// TwinCAT 3 PLC project ApicoPLC
// ProgramVersion: 3.1.4023.0
// libraries:
//   SPT Base Types, * (Beckhoff Automation LLC)
//   SPT Components, * (Beckhoff Automation LLC)
//   SPT Event Logger, * (Beckhoff Automation LLC)
//   SPT Utilities, * (Beckhoff Automation LLC)
//   Tc2_EtherCAT, * (Beckhoff Automation GmbH)
//   Tc2_Standard, * (Beckhoff Automation GmbH)
//   Tc2_System, * (Beckhoff Automation GmbH)
//   Tc3_EventLogger, * (Beckhoff Automation GmbH)
//   Tc3_Module, * (Beckhoff Automation GmbH)
//   Tc3_PackML_V2, * (Beckhoff Automation GmbH)
//   VisuDialogs, * (System)
//   VisuSymbols,newest,System
// project tree:
//   DUTs/Recipe/ ST_AxisRecipe.TcDUT (not stored), ST_PullWheelsRecipe.TcDUT (not stored), ST_SealerRecipe.TcDUT (not stored), ST_UnwindRecipe.TcDUT (not stored)
//   DUTs/ ST_Descriptor2.TcDUT (not stored), ST_PackML_Control.TcDUT (not stored), ST_PackML_Control_Simplified.TcDUT (not stored)
//   / GlobalTextList.TcGTLO, MAIN.TcPOU, PlcTask.TcTTO (not stored), VisualizationManager.TcVMO (not stored)
//   Machine/Components/Cylinder/ FB_Cylinder.TcPOU (not stored), I_Cylinder.TcIO (not stored), ST_Cylinder_Command.TcDUT (not stored), ST_Cylinder_Config.TcDUT (not stored), ST_Cylinder_HMI.TcDUT (not stored), ST_Cylinder_Status.TcDUT (not stored)
//   Machine/Components/ FB_SealBar.TcPOU (not stored)
//   Machine/EquipmentModules/ FB_PullWheel.TcPOU, FB_Unwind.TcPOU (not stored), FB_Sealer.TcPOU (not stored)
//   Machine/ FB_Machine.TcPOU
//   Machine/HMI Connections/ FB_ControlSource_HMI.TcPOU (not stored), FB_ControlSource_HMI_Machine.TcPOU
//   Machine/Templates/ FB_EquipmentModuleTemplate.TcPOU (not stored)
//   Machine/VISUs/VisuOjects/ V_MachineModule.TcVIS (not stored), V_Module.TcVIS (not stored)
//   Machine/VISUs/ V_Main.TcVIS
// real-time tasks:
//   TASK PlcTask: cycle T#10ms, priority 20, ADS port 350
// motion (NC):
//   TASK NC-Task 1 SAF: cycle T#2ms, priority 4, ADS port 501
//   TASK NC-Task 1 SVB: cycle T#10ms, priority 8, ADS port 511
//   AXIS Unwind (id 4)
//   AXIS Seal (id 5)
//   AXIS Pull 1 (id 6)
//   AXIS Pull 2 (id 7)
// variable links:
//   ApicoPLC/ApicoPLC Instance <-> NC-Task 1 SAF/Axes/Pull 1
//     PlcTask Inputs/MAIN.ApicoSeed.PullWheels.LeftPullWheel.BasicSlaveAxis._Axis.NcToPlc <-> Outputs/ToPlc
//     PlcTask Outputs/MAIN.ApicoSeed.PullWheels.LeftPullWheel.BasicSlaveAxis._Axis.PlcToNc <-> Inputs/FromPlc
//   ApicoPLC/ApicoPLC Instance <-> NC-Task 1 SAF/Axes/Pull 2
//     PlcTask Inputs/MAIN.ApicoSeed.PullWheels.RightPullWheel.BasicSlaveAxis._Axis.NcToPlc <-> Outputs/ToPlc
//     PlcTask Outputs/MAIN.ApicoSeed.PullWheels.RightPullWheel.BasicSlaveAxis._Axis.PlcToNc <-> Inputs/FromPlc
//   ApicoPLC/ApicoPLC Instance <-> NC-Task 1 SAF/Axes/Seal
//     PlcTask Inputs/MAIN.ApicoSeed.Sealer.SealerAxis.BasicAxis._Axis.NcToPlc <-> Outputs/ToPlc
//     PlcTask Outputs/MAIN.ApicoSeed.Sealer.SealerAxis.BasicAxis._Axis.PlcToNc <-> Inputs/FromPlc
//   ApicoPLC/ApicoPLC Instance <-> NC-Task 1 SAF/Axes/Unwind
//     PlcTask Inputs/MAIN.ApicoSeed.Unwind.Axis.BasicAxis._Axis.NcToPlc <-> Outputs/ToPlc
//     PlcTask Outputs/MAIN.ApicoSeed.Unwind.Axis.BasicAxis._Axis.PlcToNc <-> Inputs/FromPlc

// ---- Machine/EquipmentModules/FB_PullWheel.TcPOU
FUNCTION_BLOCK FB_PullWheel EXTENDS FB_PackML_BaseModule
VAR
    // Sub module definitions here

    // List of sub modules
    ipSubModules_Init : ARRAY[1..Parameters_PackML_Base.MAX_NO_OF_SUBMODULES] OF I_PackML_BaseModule := [];

    // Component definitions here
    LeftPullWheel     : FB_Component_BasicSlaveAxis := (Name := 'Left');
    RightPullWheel    : FB_Component_BasicSlaveAxis := (Name := 'Right');
    PullWheelCylinder : FB_Cylinder                 := (Name := 'Cylinder');

    // List of Components
    ipComponents_Init : ARRAY[1..Parameters_PackML_Base.MAX_NO_OF_COMPONENTS] OF I_ComponentBase
        := [LeftPullWheel, RightPullWheel, PullWheelCylinder];

    //Alarms for this module
    PullWheelAlarms : ARRAY[1..PULL_WHEELS_ALARM_COUNT] OF FB_TcAlarm;

	//Data for recipe
	Recipe : ST_PullWheelsRecipe;
    (*Parameters from PackTags for module
    _Param  : ARRAY[1..10] OF ST_Descriptor2;*)
    _Report : ARRAY[1..10] OF ST_Descriptor2;

    //HMI Control for EM
    fbControlSourceHMI : FB_ControlSource_HMI;
END_VAR

VAR CONSTANT

    //reports 
    FAULT : INT := 1;

    //Alarms
    PULL_WHEELS_ALARM_COUNT : INT := 5;
END_VAR

//Simulation variables for messaging
VAR
    ErrorInput : BOOL;
    WarnInput  : BOOL;
    InfoInput  : BOOL;
END_VAR

METHOD PROTECTED Aborting
VAR_INPUT
END_VAR
CASE SequenceState OF
    0:
        NoStateTasksToComplete := FALSE;
        SequenceState          := SequenceState + 10;
    10:
        LeftPullWheel.Stop();
        RightPullWheel.Stop();
        IF LeftPullWheel.Stopped AND RightPullWheel.Stopped THEN
            SequenceState := SequenceState + 10;
        END_IF
    20:
        // Disable here
        LeftPullWheel.Disable();
        RightPullWheel.Disable();
        PullWheelCylinder.Retract();

        // Check not enabled here
        IF NOT LeftPullWheel.Enabled AND NOT RightPullWheel.Enabled AND PullWheelCylinder.Retracted THEN
            SequenceState := SequenceState + 10;
        END_IF

        StateTasksComplete := TRUE;
END_CASE

SUPER^.Aborting();
END_METHOD

PROPERTY Acceleration : LREAL
SET
Recipe.LeftAxis.Acceleration := Acceleration;
Recipe.RightAxis.Acceleration := Acceleration;
END_SET
END_PROPERTY

METHOD PROTECTED Clearing
VAR_INPUT
END_VAR
CASE SequenceState OF
    0:
        NoStateTasksToComplete := FALSE;
        SequenceState          := SequenceState + 10;
    10:
        //Reset any alarms that get latched
        PullWheelAlarms[E_PullWheels.StartTimeout].Clear(0, 0);
        SequenceState := SequenceState + 10;
    20:
        // Enable here
        LeftPullWheel.Enable();
        RightPullWheel.Enable();

        // Check enabled here
        IF LeftPullWheel.Enabled AND RightPullWheel.Enabled THEN
            SequenceState := SequenceState + 10;
        END_IF
    30:
        StateTasksComplete := TRUE;
END_CASE

SUPER^.Clearing();
END_METHOD

METHOD PROTECTED CreateEvents
VAR_INPUT
END_VAR
// Add your event creation here
F_CreateAllEventsInClass(Alarms     := PullWheelAlarms,
                         ClassSize  := SIZEOF(TC_EVENTS.PullWheels),
                         pInitEvent := ADR(TC_EVENTS.PullWheels.InitReferenceEvent),
                         Prefix     := _Name);

// Super call to base
SUPER^.CreateEvents();
END_METHOD

METHOD CyclicLogic
VAR_INPUT
END_VAR
IF NOT _InitComplete THEN
    _InitComplete := Initialize();
    RETURN;
END_IF

SUPER^.CyclicLogic();

//HMI control for EM
fbControlSourceHMI.CyclicLogic();

//Set the current alarm severity for this module
_CurrentAlarmSeverity := F_GetMaxSeverityRaised(Alarms := PullWheelAlarms, CurrentSeverity := _CurrentAlarmSeverity);

//Simulate Alarm Messaging
CyclicLogic_Simulation();
END_METHOD

METHOD CyclicLogic_Simulation
VAR_INPUT
END_VAR

VAR_INST
END_VAR
(*	
This is just for testing. Real hardware can be setup in other places
Here the alarms will raise and clear on its own if the input changes	
*)

//Generic Alarms for Testing
IF ErrorInput AND NOT PullWheelAlarms[E_PullWheels.AlarmMessage].bRaised THEN
    RaiseAlarm2Args(PullWheelAlarms[E_PullWheels.AlarmMessage], '', '');
ELSIF NOT ErrorInput AND PullWheelAlarms[E_PullWheels.AlarmMessage].bRaised THEN
    PullWheelAlarms[E_PullWheels.AlarmMessage].Clear(0, 0);
END_IF

IF WarnInput AND NOT PullWheelAlarms[E_PullWheels.WarnMessage].bRaised THEN
    RaiseAlarm2Args(PullWheelAlarms[E_PullWheels.WarnMessage], '', '');
ELSIF NOT WarnInput AND PullWheelAlarms[E_PullWheels.WarnMessage].bRaised THEN
    PullWheelAlarms[E_PullWheels.WarnMessage].Clear(0, 0);
END_IF

IF InfoInput AND NOT PullWheelAlarms[E_PullWheels.InfoMessage].bRaised THEN
    RaiseAlarm2Args(PullWheelAlarms[E_PullWheels.InfoMessage], '', '');
ELSIF NOT InfoInput AND PullWheelAlarms[E_PullWheels.InfoMessage].bRaised THEN
    PullWheelAlarms[E_PullWheels.InfoMessage].Clear(0, 0);
END_IF
END_METHOD

METHOD PROTECTED Execute
VAR_INPUT
END_VAR
// Function based on mode.  NO need to make SUPER^.Executing() since it does nothing.
CASE _CurrentMode OF
    E_PMLUnitMode.ePMLUnitMode_Production:
        IF LeftPullWheel.InPosition AND NOT LeftPullWheel.Busy THEN
            PullWheelCylinder.Retract();
            IF PullWheelCylinder.Retracted THEN
                StateComplete();
            END_IF
        END_IF
    E_PMLUnitMode.ePMLUnitMode_Maintenance:
        ;
    E_PMLUnitMode.ePMLUnitMode_Manual:
        ;
END_CASE
END_METHOD

//! @summary Basic module initialization logic
METHOD PROTECTED Initialize : BOOL;
VAR
    i                        : UDINT;
    varInfo                  : __SYSTEM.VAR_INFO;
    AllSubUnitsInitialized   : BOOL := TRUE;
    AllComponentsInitialized : BOOL := TRUE;
END_VAR

//! @description This method is called by <c>CyclicLogic()</c> as required
Initialize := FALSE;
CASE DescendantSequenceState OF
    0:
        // Define the interfaces to the different subunits (Must take place before SUPER^.initialize call)
        FOR i := 1 TO SPT_BaseTypes.Parameters_PackML_Base.MAX_NO_OF_SUBMODULES DO
            ipSubModules[i] := ipSubModules_Init[i];
        END_FOR

        FOR i := 1 TO SPT_BaseTypes.Parameters_PackML_Base.MAX_NO_OF_COMPONENTS DO
            ipComponents[i] := ipComponents_Init[i];
        END_FOR

        _LogModeChanges         := FALSE;
        _LogStateChanges        := FALSE;
        DescendantSequenceState := DescendantSequenceState + 10;
    10:
        //Setup Custom modes here

        (*CustomModes(eMode                          :=,
                    sName                          :=,
                    bDisableClearing               :=,
                    bDisableStarting               :=,
                    bDisableSuspended              :=,
                    bDisableStopping               :=,
                    bDisableAborting               :=,
                    bDisableHolding                :=,
                    bDisableHeld                   :=,
                    bDisableUnholding              :=,
                    bDisableSuspending             :=,
                    bDisableUnsuspending           :=,
                    bDisableResetting              :=,
                    bDisableIdle                   :=,
                    bDisableCompleting             :=,
                    bDisableComplete               :=,
                    bEnableUnitModeChangeStopped   :=,
                    bEnableUnitModeChangeIdle      :=,
                    bEnableUnitModeChangeSuspended :=,
                    bEnableUnitModeChangeExecute   :=,
                    bEnableUnitModeChangeAborted   :=,
                    bEnableUnitModeChangeHeld      :=,
                    bEnableUnitModeChangeComplete  :=,
                    bError                         =>,
                    nErrorId                       =>);*)
        DescendantSequenceState := DescendantSequenceState + 10;
    20:
        //Copy Mode names
        FOR i := 1 TO 3 DO
            ModeNames[i] := F_UnitModeToString(UDINT_TO_DINT(i));
        END_FOR

        Initialize_TagData();
		RegisterExternalController(Controller := fbControlSourceHMI);
		fbControlSourceHMI.CyclicLogic();
        DescendantSequenceState := DescendantSequenceState + 10;
    30:
        //Call the Super
        IF SUPER^.Initialize() THEN
            DescendantSequenceState := DescendantSequenceState + 10;
        END_IF
    40:
        Initialize := TRUE;
END_CASE
END_METHOD

METHOD Initialize_TagData
VAR_INPUT
END_VAR
// Reports
_Report[FAULT].ID    := TO_DINT(1 * 10 + 1);
_Report[FAULT].Name  := 'Fault ID';
_Report[FAULT].Unit  := 'n/a';

//Recipe
Recipe.Length := 100;
Recipe.LeftAxis.Velocity := 100;
Recipe.LeftAxis.Acceleration := 1000;
Recipe.RightAxis.Velocity := 100;
Recipe.RightAxis.Acceleration := 1000;
END_METHOD

PROPERTY Length : LREAL
GET
Length := Recipe.Length;
END_GET
SET
Recipe.Length := Length;
END_SET
END_PROPERTY

METHOD RaiseAlarm2Args
VAR_IN_OUT
    Alarm : FB_TcAlarm; //Alarm to be raised
END_VAR

VAR_INPUT
    String_1 : STRING; //First String Parameter (The Name of this component will be applied first automatically)
    String_2 : STRING; //Second String Parameter
END_VAR
F_RaiseAlarmWithStringParameters(Alarm    := Alarm,
                                 String_1 := Name,
                                 String_2 := String_1,
                                 String_3 := String_2);
END_METHOD

METHOD PROTECTED Resetting
VAR_INPUT
END_VAR
CASE _CurrentMode OF
    //=================================PRODUCTION MODE==================================
    E_PMLUnitMode.ePMLUnitMode_Production:
        CASE SequenceState OF
            0:
                NoStateTasksToComplete := FALSE;
                SequenceState          := SequenceState + 10;
            10:
                /// No reason to gear to the master LeftPullWheel.Master1  REF= MAIN.ApicoSeed.Master.Axis;
                RightPullWheel.Master1 REF= LeftPullWheel.Axis;

                ///LeftPullWheel.GearIn();
                RightPullWheel.GearIn();
                SequenceState := SequenceState + 10;
            20:
                IF (*LeftPullWheel.InGear AND*) RightPullWheel.InGear THEN
                    StateTasksComplete := TRUE;
                END_IF
        END_CASE

    //=================================MAINTENANCE & MANUAL MODE==================================	
    E_PMLUnitMode.ePMLUnitMode_Maintenance, E_PMLUnitMode.ePMLUnitMode_Manual:
        ;
END_CASE

SUPER^.Resetting();
END_METHOD

METHOD PROTECTED Starting
VAR_INPUT
END_VAR

VAR_INST
    StartTimer : TON;
END_VAR
CASE _CurrentMode OF
    //=================================PRODUCTION MODE==================================
    E_PMLUnitMode.ePMLUnitMode_Production:
        CASE SequenceState OF
            0:
                // Delay 1 scan to make sure timer is off.  Not guarnteed from last time where it finished.
                NoStateTasksToComplete := FALSE;
                SequenceState          := SequenceState + 10;
            10:
                PullWheelCylinder.Extend();
                IF PullWheelCylinder.Extended THEN
                    NoStateTasksToComplete     := FALSE;
                    LeftPullWheel.Velocity     := Recipe.LeftAxis.Velocity;
                    LeftPullWheel.Acceleration := Recipe.LeftAxis.Acceleration;
                    LeftPullWheel.MoveRelative(Distance := Recipe.Length, FALSE);
                    SequenceState := SequenceState + 10;
                END_IF
            20:
                IF LeftPullWheel.Busy THEN
                    SequenceState := SequenceState + 10;
                END_IF

                IF StartTimer.Q AND NOT PullWheelAlarms[E_PullWheels.StartTimeout].bRaised THEN
                    RaiseAlarm2Args(PullWheelAlarms[E_PullWheels.StartTimeout], '', '');
                    SequenceState := SequenceState + 10;
                END_IF
            30:
                StateTasksComplete := TRUE;
        END_CASE

    //=================================MAINTENANCE & MANUAL MODE==================================
    E_PMLUnitMode.ePMLUnitMode_Maintenance, E_PMLUnitMode.ePMLUnitMode_Manual:
        ;
END_CASE

SUPER^.Starting();
StartTimer(IN := ((SequenceState = 10) OR (SequenceState = 20)), PT := T#3S);
END_METHOD

METHOD PROTECTED Stopping
VAR_INPUT
END_VAR
CASE _CurrentMode OF
    //=================================PRODUCTION MODE==================================
    E_PMLUnitMode.ePMLUnitMode_Production:
        CASE SequenceState OF
            0:
                NoStateTasksToComplete := FALSE;
                PullWheelCylinder.Retract();
                SequenceState := SequenceState + 10;
            10:
                IF PullWheelCylinder.Retracted THEN
                    SequenceState := SequenceState + 10;
                END_IF
            20:
                StateTasksComplete := TRUE;
        END_CASE

    //=================================MAINTENANCE & MANUAL MODE==================================
    E_PMLUnitMode.ePMLUnitMode_Maintenance, E_PMLUnitMode.ePMLUnitMode_Manual:
        ;
END_CASE

SUPER^.Stopping();
END_METHOD

PROPERTY Velocity : LREAL
SET
Recipe.LeftAxis.Velocity := Velocity;
Recipe.RightAxis.Velocity := Velocity;
END_SET
END_PROPERTY

END_FUNCTION_BLOCK

// ---- Machine/FB_Machine.TcPOU
FUNCTION_BLOCK FB_Machine EXTENDS FB_PackML_BaseModule // IMPLEMENTS I_ControlsProductionRate
VAR
    // Sub Modules
    PullWheels : FB_PullWheel := (Name := 'Pull Wheel', LogStateChanges := TRUE);
    Sealer     : FB_Sealer    := (Name := 'Sealer', LogStateChanges := TRUE);
    Unwind     : FB_Unwind    := (Name := 'Unwind', LogStateChanges := TRUE);

    //Initial List of SubModules
    ipSubModules_Init :
        ARRAY[1..Parameters_PackML_Base.MAX_NO_OF_SUBMODULES] OF I_PackML_BaseModule := [PullWheels, Sealer, Unwind];

    // Components

    //Initial List of Components
    ipComponents_Init : ARRAY[1..Parameters_PackML_Base.MAX_NO_OF_COMPONENTS] OF I_ComponentBase := [];

    //Alarms for this module
    MachineAlarms : ARRAY[1..MACHINE_ALARM_COUNT] OF FB_TcAlarm;
	
	//Current Recipe Name
	CurrentRecipeName : STRING;

    //Get Data From PackML? Else RecipeManager is running
    DataFromPackML : BOOL := TRUE;

    //Data 
    sealTimeStart : ULINT;
    sealTimeEnd   : ULINT;
    sealingTime   : LREAL;
    sealTrig      : R_TRIG;
    pullTimeStart : ULINT;
    pullTimeEnd   : ULINT;
    pullingTime   : LREAL;
    pulltrig      : R_TRIG;
    partTimeStart : ULINT;
    partTimeEnd   : ULINT;
    partTime      : LREAL;
    parts         : DINT;
    product       : DINT;

    //Pack Tags for System
    {attribute 'OPC.UA.DA' := '1'}
    _PackTags : ST_PackMLv30Ext; //ST_PackMLv30 is obsolete in Tc3_PackML_V2
END_VAR

VAR CONSTANT
    //PackTag parameter IDs
    LENGTH         : INT := 1;
    SEALTEMP       : INT := 2;
    SEALTIME       : INT := 3;
    PULLWHEELS_VEL : INT := 4;
    PULLWHEELS_ACC : INT := 5;
    SEALER_VEL     : INT := 6;
    SEALER_ACC     : INT := 7;
    UNWIND_VEL     : INT := 8;
    UNWIND_ACC     : INT := 9;
    OPEN_POS       : INT := 10;
    CLOSED_POS     : INT := 11;

    //Alarm count constant
    MACHINE_ALARM_COUNT : INT := 6;
END_VAR

// Simulation variables
VAR
    EstopInput  : BOOL;
    KurwaJebanaInput : BOOL;
    ErrorInput  : BOOL;
    WarnInput   : BOOL;
    InfoInput   : BOOL;
END_VAR

METHOD PROTECTED Completing
VAR_INPUT
END_VAR
CASE _CurrentMode OF
    //=================================PRODUCTION MODE==================================
    E_PMLUnitMode.ePMLUnitMode_Production:
        StateComplete();
    E_PMLUnitMode.ePMLUnitMode_Maintenance, E_PMLUnitMode.ePMLUnitMode_Manual:
        SUPER^.Completing();
END_CASE
END_METHOD

METHOD PROTECTED CreateEvents
VAR_INPUT
END_VAR
// Add your event creation here
F_CreateAllEventsInClass(Alarms     := MachineAlarms,
                         ClassSize  := SIZEOF(TC_Events.ApicoSeed),
                         pInitEvent := ADR(TC_EVENTS.ApicoSeed.InitReferenceEvent),
                         Prefix     := Name);

// Super call to base
SUPER^.CreateEvents();
END_METHOD

METHOD CyclicLogic
VAR_INPUT
END_VAR
IF NOT _InitComplete THEN
    _InitComplete := Initialize();
    RETURN;
END_IF

SUPER^.CyclicLogic();

// Fill in the PackTags for the machine output
_PackTags.Status.StateCurrent    := _CurrentState;
_PackTags.Status.UnitModeCurrent := _CurrentMode;
UpdateModeTimers();

//This is just to simulate some IO for alarms
CyclicLogic_Simulation();
END_METHOD

METHOD CyclicLogic_Simulation
VAR_INPUT
END_VAR

VAR_INST
END_VAR
(*	
This is just for testing. Real hardware can be setup in other places
Here the alarms will raise and clear on its own if the input changes	
*)
IF EstopInput AND NOT MachineAlarms[E_ApicoSeed.EmergencyStop].bRaised THEN
    RaiseAlarm2Args(MachineAlarms[E_ApicoSeed.EmergencyStop], '', '');
ELSIF NOT EstopInput AND MachineAlarms[E_ApicoSeed.EmergencyStop].bRaised THEN
    MachineAlarms[E_ApicoSeed.EmergencyStop].Clear(0, 0);
END_IF

IF KurwaJebanaInput AND NOT MachineAlarms[E_ApicoSeed.KurwaJebana].bRaised THEN
    RaiseAlarm2Args(MachineAlarms[E_ApicoSeed.KurwaJebana], '', '');
ELSIF NOT KurwaJebanaInput AND MachineAlarms[E_ApicoSeed.KurwaJebana].bRaised THEN
    MachineAlarms[E_ApicoSeed.KurwaJebana].Clear(0, 0);
END_IF

//Generic Alarms for Testing
IF ErrorInput AND NOT MachineAlarms[E_ApicoSeed.AlarmMessage].bRaised THEN
    RaiseAlarm2Args(MachineAlarms[E_ApicoSeed.AlarmMessage], '', '');
ELSIF NOT ErrorInput AND MachineAlarms[E_ApicoSeed.AlarmMessage].bRaised THEN
    MachineAlarms[E_ApicoSeed.AlarmMessage].Clear(0, 0);
END_IF

IF WarnInput AND NOT MachineAlarms[E_ApicoSeed.WarnMessage].bRaised THEN
    RaiseAlarm2Args(MachineAlarms[E_ApicoSeed.WarnMessage], '', '');
ELSIF NOT WarnInput AND MachineAlarms[E_ApicoSeed.WarnMessage].bRaised THEN
    MachineAlarms[E_ApicoSeed.WarnMessage].Clear(0, 0);
END_IF

IF InfoInput AND NOT MachineAlarms[E_ApicoSeed.InfoMessage].bRaised THEN
    RaiseAlarm2Args(MachineAlarms[E_ApicoSeed.InfoMessage], '', '');
ELSIF NOT InfoInput AND MachineAlarms[E_ApicoSeed.InfoMessage].bRaised THEN
    MachineAlarms[E_ApicoSeed.InfoMessage].Clear(0, 0);
END_IF
END_METHOD

METHOD PROTECTED FINAL Execute
VAR_INPUT
END_VAR
CASE _CurrentMode OF
    //=================================PRODUCTION MODE==================================
    E_PMLUnitMode.ePMLUnitMode_Production:
        (* Run the sequence to make products 
		 Unwind Runs Slowly 
		 Pull Wheels Run 
		 Jaws Seal, and Repeat until production reached*)
        sealTrig(CLK := SequenceState = 10);
        IF sealTrig.Q THEN
            partTimeStart := F_GetActualDcTime64();
            sealTimeStart := partTimeStart;
        END_IF

        pulltrig(CLK := SequenceState = 20);
        IF pulltrig.Q THEN
            pullTimeStart := F_GetActualDcTime64();
        END_IF

		IF THIS^.Sealer.sealbar.InTempRange THEN
			CASE SequenceState OF
				0: //Started
					Unwind.ChangeState(E_PMLCommand.ePMLCommand_Start);
					IF Unwind.CurrentState = E_PMLState.ePMLState_Execute THEN
						SequenceState := SequenceState + 10;
					END_IF
				10: // SEAL First
					Sealer.ChangeState(E_PMLCommand.ePMLCommand_Start);
					IF Sealer.CurrentState = E_PMLState.ePMLState_Complete THEN
						Sealer.ChangeState(E_PMLCommand.ePMLCommand_Reset);
						SequenceState := SequenceState + 10;
						SealTimeEnd   := F_GetActualDcTime64();
						sealingTime   := ULINT_TO_LREAL(sealtimeEnd - sealTimeStart) * 1E-9;
					END_IF
				20: // Run Pullwheels
					PullWheels.ChangeState(E_PMLCommand.ePMLCommand_Start);
					IF PullWheels.CurrentState = E_PMLState.ePMLState_Complete THEN
						partTimeEnd   := F_GetActualDcTime64();
						parts         := parts + 1;
						SequenceState := 10;
						PullWheels.ChangeState(E_PMLCommand.ePMLCommand_Reset);
						pullTimeEnd := F_GetActualDcTime64();
						pullingTime := ULINT_TO_LREAL(pullTimeEnd - pullTimeStart) * 1E-9;
					END_IF
			END_CASE
		ELSE
			ChangeState(E_PMLCommand.ePMLCommand_Suspend);
		END_IF
			
    //=================================MAINTENANCE MODE==================================	
    E_PMLUnitMode.ePMLUnitMode_Maintenance:
        ;

    //=================================MANUAL MODE==================================
    E_PMLUnitMode.ePMLUnitMode_Manual:
        ;
END_CASE
END_METHOD

METHOD PROTECTED Held
VAR_INPUT
END_VAR
END_METHOD

METHOD PROTECTED HMIPermissions
VAR_INPUT
END_VAR
//General Mode Based Monitoring and handling of HMI control
CASE _CurrentMode OF
    E_PMLUnitMode.ePMLUnitMode_Production:
        CASE _CurrentState OF
            E_PMLState.ePMLState_Stopped:
                AllowHMIControl(ThisModuleOnly := TRUE); //Allow control for recovery
            E_PMLState.ePMLState_Idle:
                //BlockHMIControl();
				AllowHMIControl(ThisModuleOnly := TRUE); //Allow control for recovery
            E_PMLState.ePMLState_Suspended:
                BlockHMIControl();
            E_PMLState.ePMLState_Execute:
                BlockHMIControl();
            E_PMLState.ePMLState_Aborted:
                AllowHMIControl(ThisModuleOnly := TRUE); //Allow control for recovery
            E_PMLState.ePMLState_Held:
                AllowHMIControl(ThisModuleOnly := TRUE); //Allow control for recovery
            E_PMLState.ePMLState_Complete:
                BlockHMIControl();
        END_CASE
		
        //AllowHMIControl(ThisModuleOnly := FALSE);
    E_PMLUnitMode.ePMLUnitMode_Manual:
        AllowHMIControl(ThisModuleOnly := FALSE);
    E_PMLUnitMode.ePMLUnitMode_Maintenance:
        AllowHMIControl(ThisModuleOnly := FALSE);
END_CASE
END_METHOD

METHOD PROTECTED HoldImmediate
VAR_INPUT
END_VAR
ChangeState(E_PMLCommand.ePMLCommand_Hold);
END_METHOD

METHOD PROTECTED Holding
VAR_INPUT
END_VAR
CASE _CurrentMode OF
    //=================================PRODUCTION MODE==================================
    E_PMLUnitMode.ePMLUnitMode_Production:
        IF (Sealer.CurrentState = E_PMLState.ePMLState_Complete OR Sealer.CurrentState = E_PMLState.ePMLState_Idle) AND
           (PullWheels.CurrentState = E_PMLState.ePMLState_Complete OR PullWheels.CurrentState = E_PMLState.ePMLState_Idle) THEN
            StateComplete();
        END_IF
    E_PMLUnitMode.ePMLUnitMode_Maintenance, E_PMLUnitMode.ePMLUnitMode_Manual:
        SUPER^.Holding();
END_CASE
END_METHOD

METHOD PROTECTED Initialize : BOOL
VAR
    i : UDINT; //Generic iteration value
END_VAR
Initialize := FALSE;
CASE DescendantSequenceState OF
    0:
        // Define the interfaces to the different subunits (Must take place before SUPER^.initialize call)
        FOR i := 1 TO SPT_BaseTypes.Parameters_PackML_Base.MAX_NO_OF_SUBMODULES DO
            ipSubModules[i] := ipSubModules_Init[i];
        END_FOR

        FOR i := 1 TO SPT_BaseTypes.Parameters_PackML_Base.MAX_NO_OF_COMPONENTS DO
            ipComponents[i] := ipComponents_Init[i];
        END_FOR

        _LogModeChanges         := FALSE;
        _LogStateChanges        := FALSE;
        DescendantSequenceState := DescendantSequenceState + 10;
    10:
        //Setup Custom modes here

        (*CustomModes(eMode                          :=,
                    sName                          :=,
                    bDisableClearing               :=,
                    bDisableStarting               :=,
                    bDisableSuspended              :=,
                    bDisableStopping               :=,
                    bDisableAborting               :=,
                    bDisableHolding                :=,
                    bDisableHeld                   :=,
                    bDisableUnholding              :=,
                    bDisableSuspending             :=,
                    bDisableUnsuspending           :=,
                    bDisableResetting              :=,
                    bDisableIdle                   :=,
                    bDisableCompleting             :=,
                    bDisableComplete               :=,
                    bEnableUnitModeChangeStopped   :=,
                    bEnableUnitModeChangeIdle      :=,
                    bEnableUnitModeChangeSuspended :=,
                    bEnableUnitModeChangeExecute   :=,
                    bEnableUnitModeChangeAborted   :=,
                    bEnableUnitModeChangeHeld      :=,
                    bEnableUnitModeChangeComplete  :=,
                    bError                         =>,
                    nErrorId                       =>);*)
        DescendantSequenceState := DescendantSequenceState + 10;
    20:
        //Copy Mode names
        FOR i := 1 TO 3 DO
            ModeNames[i] := F_UnitModeToString(UDINT_TO_DINT(i));
        END_FOR

        DescendantSequenceState := DescendantSequenceState + 10;
    30:
        // Initialize Recipes 
        Initialize_Recipes();
        DescendantSequenceState := DescendantSequenceState + 10;
    40:
        //Call the Super
        IF SUPER^.Initialize() THEN
            DescendantSequenceState := DescendantSequenceState + 10;
        END_IF
    50:
        Initialize := TRUE;
END_CASE
END_METHOD

METHOD Initialize_Recipes
VAR_INPUT
END_VAR
// configuration of parameters Max Speed
_packTags.Command.Parameter[1].ID    := 1;
_packTags.Command.Parameter[1].Name  := 'Max Speed';
_packTags.Command.Parameter[1].Unit  := '/min';
_packTags.Command.Parameter[1].Value := 180;
_packTags.Command.Parameter[2].ID    := 2;
_packTags.Command.Parameter[2].Name  := 'Product to Run';
_packTags.Command.Parameter[2].Unit  := '';
_packTags.Command.Parameter[2].Value := 1;

// Recipe Product 1
_PackTags.Command.Product[1].ProductID                              := 100;
_PackTags.Command.Product[1].Ingredients[1].IngredientID            := 1;
_PackTags.Command.Product[1].Ingredients[1].Parameter[1].ID         := _PackTags.Command.Product[1].ProductID * 10 + 1;
_PackTags.Command.Product[1].Ingredients[1].Parameter[1].Name       := 'Material Type';
_PackTags.Command.Product[1].Ingredients[1].Parameter[1].Unit       := 'n/a';
_PackTags.Command.Product[1].Ingredients[1].Parameter[1].Value      := 5;
_PackTags.Command.Product[1].Ingredients[1].Parameter[2].ID         := _PackTags.Command.Product[1].ProductID * 10 + 2;
_PackTags.Command.Product[1].Ingredients[1].Parameter[2].Name       := 'Material Thickness';
_PackTags.Command.Product[1].Ingredients[1].Parameter[2].Unit       := 'um';
_PackTags.Command.Product[1].Ingredients[1].Parameter[2].Value      := 240;
_PackTags.Command.Product[1].ProcessVariables[LENGTH].ID            := _PackTags.Command.Product[1].ProductID * 20 + 1;
_PackTags.Command.Product[1].ProcessVariables[LENGTH].Name          := 'Length';
_PackTags.Command.Product[1].ProcessVariables[LENGTH].Unit          := 'mm';
_PackTags.Command.Product[1].ProcessVariables[LENGTH].Value         := 100;
_PackTags.Command.Product[1].ProcessVariables[SEALTEMP].ID          := _PackTags.Command.Product[1].ProductID * 20 + 2;
_PackTags.Command.Product[1].ProcessVariables[SEALTEMP].Name        := 'Sealing Temp';
_PackTags.Command.Product[1].ProcessVariables[SEALTEMP].Unit        := 'C';
_PackTags.Command.Product[1].ProcessVariables[SEALTEMP].Value       := 100;
_PackTags.Command.Product[1].ProcessVariables[SEALTIME].ID          := _PackTags.Command.Product[1].ProductID * 20 + 3;
_PackTags.Command.Product[1].ProcessVariables[SEALTIME].Name        := 'Sealing Time';
_PackTags.Command.Product[1].ProcessVariables[SEALTIME].Unit        := 'ms';
_PackTags.Command.Product[1].ProcessVariables[SEALTIME].Value       := 50;
_PackTags.Command.Product[1].ProcessVariables[PULLWHEELS_VEL].ID    := _PackTags.Command.Product[1].ProductID * 20 + 4;
_PackTags.Command.Product[1].ProcessVariables[PULLWHEELS_VEL].Name  := 'Pull Wheels Vel';
_PackTags.Command.Product[1].ProcessVariables[PULLWHEELS_VEL].Unit  := 'mm/s';
_PackTags.Command.Product[1].ProcessVariables[PULLWHEELS_VEL].Value := 100;
_PackTags.Command.Product[1].ProcessVariables[PULLWHEELS_ACC].ID    := _PackTags.Command.Product[1].ProductID * 20 + 5;
_PackTags.Command.Product[1].ProcessVariables[PULLWHEELS_ACC].Name  := 'Pull Wheels Acc';
_PackTags.Command.Product[1].ProcessVariables[PULLWHEELS_ACC].Unit  := 'mm/s2';
_PackTags.Command.Product[1].ProcessVariables[PULLWHEELS_ACC].Value := 1000;
_PackTags.Command.Product[1].ProcessVariables[OPEN_POS].ID          := _PackTags.Command.Product[1].ProductID * 20 + 6;
_PackTags.Command.Product[1].ProcessVariables[OPEN_POS].Name        := 'Sealer Open Position';
_PackTags.Command.Product[1].ProcessVariables[OPEN_POS].Unit        := 'mm';
_PackTags.Command.Product[1].ProcessVariables[OPEN_POS].Value       := 105;
_PackTags.Command.Product[1].ProcessVariables[CLOSED_POS].ID        := _PackTags.Command.Product[1].ProductID * 20 + 7;
_PackTags.Command.Product[1].ProcessVariables[CLOSED_POS].Name      := 'Sealer Closed Position';
_PackTags.Command.Product[1].ProcessVariables[CLOSED_POS].Unit      := 'mm';
_PackTags.Command.Product[1].ProcessVariables[CLOSED_POS].Value     := 250;
_PackTags.Command.Product[1].ProcessVariables[SEALER_VEL].ID        := _PackTags.Command.Product[1].ProductID * 20 + 8;
_PackTags.Command.Product[1].ProcessVariables[SEALER_VEL].Name      := 'Sealer Vel';
_PackTags.Command.Product[1].ProcessVariables[SEALER_VEL].Unit      := 'mm/s';
_PackTags.Command.Product[1].ProcessVariables[SEALER_VEL].Value     := 100;
_PackTags.Command.Product[1].ProcessVariables[SEALER_ACC].ID        := _PackTags.Command.Product[1].ProductID * 20 + 9;
_PackTags.Command.Product[1].ProcessVariables[SEALER_ACC].Name      := 'Sealer Acc';
_PackTags.Command.Product[1].ProcessVariables[SEALER_ACC].Unit      := 'mm/s2';
_PackTags.Command.Product[1].ProcessVariables[SEALER_ACC].Value     := 1000;
_PackTags.Command.Product[1].ProcessVariables[UNWIND_VEL].ID        := _PackTags.Command.Product[1].ProductID * 20 + 10;
_PackTags.Command.Product[1].ProcessVariables[UNWIND_VEL].Name      := 'Unwind Vel';
_PackTags.Command.Product[1].ProcessVariables[UNWIND_VEL].Unit      := 'mm/s';
_PackTags.Command.Product[1].ProcessVariables[UNWIND_VEL].Value     := 100;
_PackTags.Command.Product[1].ProcessVariables[UNWIND_ACC].ID        := _PackTags.Command.Product[1].ProductID * 20 + 11;
_PackTags.Command.Product[1].ProcessVariables[UNWIND_ACC].Name      := 'Unwind Acc';
_PackTags.Command.Product[1].ProcessVariables[UNWIND_ACC].Unit      := 'mm/s2';
_PackTags.Command.Product[1].ProcessVariables[UNWIND_ACC].Value     := 1000;

// Product 2
_PackTags.Command.Product[2].ProductID                         := 100;
_PackTags.Command.Product[2].Ingredients[1].IngredientID       := 1;
_PackTags.Command.Product[2].Ingredients[1].Parameter[1].ID    := _PackTags.Command.Product[1].ProductID * 10 + 1;
_PackTags.Command.Product[2].Ingredients[1].Parameter[1].Name  := 'Material Type';
_PackTags.Command.Product[2].Ingredients[1].Parameter[1].Unit  := 'n/a';
_PackTags.Command.Product[2].Ingredients[1].Parameter[1].Value := 2;
_PackTags.Command.Product[2].Ingredients[1].Parameter[2].ID    := _PackTags.Command.Product[1].ProductID * 10 + 2;
_PackTags.Command.Product[2].Ingredients[1].Parameter[2].Name  := 'Material Thickness';
_PackTags.Command.Product[2].Ingredients[1].Parameter[2].Unit  := 'um';
_PackTags.Command.Product[2].Ingredients[1].Parameter[2].Value := 220;
_PackTags.Command.Product[2].ProcessVariables[LENGTH].ID       := _PackTags.Command.Product[1].ProductID * 20 + 1;
_PackTags.Command.Product[2].ProcessVariables[LENGTH].Name     := 'Length';
_PackTags.Command.Product[2].ProcessVariables[LENGTH].Unit     := 'mm';
_PackTags.Command.Product[2].ProcessVariables[LENGTH].Value    := 55;
_PackTags.Command.Product[2].ProcessVariables[SEALTEMP].ID     := _PackTags.Command.Product[1].ProductID * 20 + 2;
_PackTags.Command.Product[2].ProcessVariables[SEALTEMP].Name   := 'Sealing Temp';
_PackTags.Command.Product[2].ProcessVariables[SEALTEMP].Unit   := 'C';
_PackTags.Command.Product[2].ProcessVariables[SEALTEMP].Value  := 110;
_PackTags.Command.Product[2].ProcessVariables[SEALTIME].ID     := _PackTags.Command.Product[1].ProductID * 20 + 3;
_PackTags.Command.Product[2].ProcessVariables[SEALTIME].Name   := 'Sealing Time';
_PackTags.Command.Product[2].ProcessVariables[SEALTIME].Unit   := 'ms';
_PackTags.Command.Product[2].ProcessVariables[SEALTIME].Value  := 100;
_PackTags.Command.Product[2].ProcessVariables[PULLWHEELS_VEL].ID    := _PackTags.Command.Product[1].ProductID * 20 + 4;
_PackTags.Command.Product[2].ProcessVariables[PULLWHEELS_VEL].Name  := 'Pull Wheels Vel';
_PackTags.Command.Product[2].ProcessVariables[PULLWHEELS_VEL].Unit  := 'mm/s';
_PackTags.Command.Product[2].ProcessVariables[PULLWHEELS_VEL].Value := 200;
_PackTags.Command.Product[2].ProcessVariables[PULLWHEELS_ACC].ID    := _PackTags.Command.Product[1].ProductID * 20 + 5;
_PackTags.Command.Product[2].ProcessVariables[PULLWHEELS_ACC].Name  := 'Pull Wheels Acc';
_PackTags.Command.Product[2].ProcessVariables[PULLWHEELS_ACC].Unit  := 'mm/s2';
_PackTags.Command.Product[2].ProcessVariables[PULLWHEELS_ACC].Value := 2000;
_PackTags.Command.Product[2].ProcessVariables[OPEN_POS].ID          := _PackTags.Command.Product[1].ProductID * 20 + 6;
_PackTags.Command.Product[2].ProcessVariables[OPEN_POS].Name        := 'Sealer Open Position';
_PackTags.Command.Product[2].ProcessVariables[OPEN_POS].Unit        := 'mm';
_PackTags.Command.Product[2].ProcessVariables[OPEN_POS].Value       := 60;
_PackTags.Command.Product[2].ProcessVariables[CLOSED_POS].ID        := _PackTags.Command.Product[1].ProductID * 20 + 7;
_PackTags.Command.Product[2].ProcessVariables[CLOSED_POS].Name      := 'Sealer Closed Position';
_PackTags.Command.Product[2].ProcessVariables[CLOSED_POS].Unit      := 'mm';
_PackTags.Command.Product[2].ProcessVariables[CLOSED_POS].Value     := 253;
_PackTags.Command.Product[2].ProcessVariables[SEALER_VEL].ID        := _PackTags.Command.Product[1].ProductID * 20 + 8;
_PackTags.Command.Product[2].ProcessVariables[SEALER_VEL].Name      := 'Sealer Vel';
_PackTags.Command.Product[2].ProcessVariables[SEALER_VEL].Unit      := 'mm/s';
_PackTags.Command.Product[2].ProcessVariables[SEALER_VEL].Value     := 200;
_PackTags.Command.Product[2].ProcessVariables[SEALER_ACC].ID        := _PackTags.Command.Product[1].ProductID * 20 + 9;
_PackTags.Command.Product[2].ProcessVariables[SEALER_ACC].Name      := 'Sealer Acc';
_PackTags.Command.Product[2].ProcessVariables[SEALER_ACC].Unit      := 'mm/s2';
_PackTags.Command.Product[2].ProcessVariables[SEALER_ACC].Value     := 2000;
_PackTags.Command.Product[2].ProcessVariables[UNWIND_VEL].ID        := _PackTags.Command.Product[1].ProductID * 20 + 10;
_PackTags.Command.Product[2].ProcessVariables[UNWIND_VEL].Name      := 'Unwind Vel';
_PackTags.Command.Product[2].ProcessVariables[UNWIND_VEL].Unit      := 'mm/s';
_PackTags.Command.Product[2].ProcessVariables[UNWIND_VEL].Value     := 200;
_PackTags.Command.Product[2].ProcessVariables[UNWIND_ACC].ID        := _PackTags.Command.Product[1].ProductID * 20 + 11;
_PackTags.Command.Product[2].ProcessVariables[UNWIND_ACC].Name      := 'Unwind Acc';
_PackTags.Command.Product[2].ProcessVariables[UNWIND_ACC].Unit      := 'mm/s2';
_PackTags.Command.Product[2].ProcessVariables[UNWIND_ACC].Value     := 2000;

//Product 3
_PackTags.Command.Product[3].ProductID                         := 307;
_PackTags.Command.Product[3].Ingredients[1].IngredientID       := 1;
_PackTags.Command.Product[3].Ingredients[1].Parameter[1].ID    := _PackTags.Command.Product[1].ProductID * 10 + 1;
_PackTags.Command.Product[3].Ingredients[1].Parameter[1].Name  := 'Material Type';
_PackTags.Command.Product[3].Ingredients[1].Parameter[1].Unit  := 'n/a';
_PackTags.Command.Product[3].Ingredients[1].Parameter[1].Value := 2;
_PackTags.Command.Product[3].Ingredients[1].Parameter[2].ID    := _PackTags.Command.Product[1].ProductID * 10 + 2;
_PackTags.Command.Product[3].Ingredients[1].Parameter[2].Name  := 'Material Thickness';
_PackTags.Command.Product[3].Ingredients[1].Parameter[2].Unit  := 'um';
_PackTags.Command.Product[3].Ingredients[1].Parameter[2].Value := 220;
_PackTags.Command.Product[3].ProcessVariables[LENGTH].ID       := _PackTags.Command.Product[1].ProductID * 20 + 1;
_PackTags.Command.Product[3].ProcessVariables[LENGTH].Name     := 'Length';
_PackTags.Command.Product[3].ProcessVariables[LENGTH].Unit     := 'mm';
_PackTags.Command.Product[3].ProcessVariables[LENGTH].Value    := 85;
_PackTags.Command.Product[3].ProcessVariables[SEALTEMP].ID     := _PackTags.Command.Product[1].ProductID * 20 + 2;
_PackTags.Command.Product[3].ProcessVariables[SEALTEMP].Name   := 'Sealing Temp';
_PackTags.Command.Product[3].ProcessVariables[SEALTEMP].Unit   := 'C';
_PackTags.Command.Product[3].ProcessVariables[SEALTEMP].Value  := 95;
_PackTags.Command.Product[3].ProcessVariables[SEALTIME].ID     := _PackTags.Command.Product[1].ProductID * 20 + 3;
_PackTags.Command.Product[3].ProcessVariables[SEALTIME].Name   := 'Sealing Time';
_PackTags.Command.Product[3].ProcessVariables[SEALTIME].Unit   := 'ms';
_PackTags.Command.Product[3].ProcessVariables[SEALTIME].Value  := 20;
_PackTags.Command.Product[3].ProcessVariables[PULLWHEELS_VEL].ID    := _PackTags.Command.Product[1].ProductID * 20 + 4;
_PackTags.Command.Product[3].ProcessVariables[PULLWHEELS_VEL].Name  := 'Pull Wheels Vel';
_PackTags.Command.Product[3].ProcessVariables[PULLWHEELS_VEL].Unit  := 'mm/s';
_PackTags.Command.Product[3].ProcessVariables[PULLWHEELS_VEL].Value := 300;
_PackTags.Command.Product[3].ProcessVariables[PULLWHEELS_ACC].ID    := _PackTags.Command.Product[1].ProductID * 20 + 5;
_PackTags.Command.Product[3].ProcessVariables[PULLWHEELS_ACC].Name  := 'Pull Wheels Acc';
_PackTags.Command.Product[3].ProcessVariables[PULLWHEELS_ACC].Unit  := 'mm/s2';
_PackTags.Command.Product[3].ProcessVariables[PULLWHEELS_ACC].Value := 3000;
_PackTags.Command.Product[3].ProcessVariables[OPEN_POS].ID          := _PackTags.Command.Product[1].ProductID * 20 + 6;
_PackTags.Command.Product[3].ProcessVariables[OPEN_POS].Name        := 'Sealer Open Position';
_PackTags.Command.Product[3].ProcessVariables[OPEN_POS].Unit        := 'mm';
_PackTags.Command.Product[3].ProcessVariables[OPEN_POS].Value       := 56;
_PackTags.Command.Product[3].ProcessVariables[CLOSED_POS].ID        := _PackTags.Command.Product[1].ProductID * 20 + 7;
_PackTags.Command.Product[3].ProcessVariables[CLOSED_POS].Name      := 'Sealer Closed Position';
_PackTags.Command.Product[3].ProcessVariables[CLOSED_POS].Unit      := 'mm';
_PackTags.Command.Product[3].ProcessVariables[CLOSED_POS].Value     := 265;
_PackTags.Command.Product[3].ProcessVariables[SEALER_VEL].ID        := _PackTags.Command.Product[1].ProductID * 20 + 8;
_PackTags.Command.Product[3].ProcessVariables[SEALER_VEL].Name      := 'Sealer Vel';
_PackTags.Command.Product[3].ProcessVariables[SEALER_VEL].Unit      := 'mm/s';
_PackTags.Command.Product[3].ProcessVariables[SEALER_VEL].Value     := 300;
_PackTags.Command.Product[3].ProcessVariables[SEALER_ACC].ID        := _PackTags.Command.Product[1].ProductID * 20 + 9;
_PackTags.Command.Product[3].ProcessVariables[SEALER_ACC].Name      := 'Sealer Acc';
_PackTags.Command.Product[3].ProcessVariables[SEALER_ACC].Unit      := 'mm/s2';
_PackTags.Command.Product[3].ProcessVariables[SEALER_ACC].Value     := 3000;
_PackTags.Command.Product[3].ProcessVariables[UNWIND_VEL].ID        := _PackTags.Command.Product[1].ProductID * 20 + 10;
_PackTags.Command.Product[3].ProcessVariables[UNWIND_VEL].Name      := 'Unwind Vel';
_PackTags.Command.Product[3].ProcessVariables[UNWIND_VEL].Unit      := 'mm/s';
_PackTags.Command.Product[3].ProcessVariables[UNWIND_VEL].Value     := 300;
_PackTags.Command.Product[3].ProcessVariables[UNWIND_ACC].ID        := _PackTags.Command.Product[1].ProductID * 20 + 11;
_PackTags.Command.Product[3].ProcessVariables[UNWIND_ACC].Name      := 'Unwind Acc';
_PackTags.Command.Product[3].ProcessVariables[UNWIND_ACC].Unit      := 'mm/s2';
_PackTags.Command.Product[3].ProcessVariables[UNWIND_ACC].Value     := 3000;

//Product 4
_PackTags.Command.Product[4].ProductID                         := 401;
_PackTags.Command.Product[4].Ingredients[1].IngredientID       := 1;
_PackTags.Command.Product[4].Ingredients[1].Parameter[1].ID    := _PackTags.Command.Product[1].ProductID * 10 + 1;
_PackTags.Command.Product[4].Ingredients[1].Parameter[1].Name  := 'Material Type';
_PackTags.Command.Product[4].Ingredients[1].Parameter[1].Unit  := 'n/a';
_PackTags.Command.Product[4].Ingredients[1].Parameter[1].Value := 2;
_PackTags.Command.Product[4].Ingredients[1].Parameter[2].ID    := _PackTags.Command.Product[1].ProductID * 10 + 2;
_PackTags.Command.Product[4].Ingredients[1].Parameter[2].Name  := 'Material Thickness';
_PackTags.Command.Product[4].Ingredients[1].Parameter[2].Unit  := 'um';
_PackTags.Command.Product[4].Ingredients[1].Parameter[2].Value := 220;
_PackTags.Command.Product[4].ProcessVariables[LENGTH].ID       := _PackTags.Command.Product[1].ProductID * 20 + 1;
_PackTags.Command.Product[4].ProcessVariables[LENGTH].Name     := 'Length';
_PackTags.Command.Product[4].ProcessVariables[LENGTH].Unit     := 'mm';
_PackTags.Command.Product[4].ProcessVariables[LENGTH].Value    := 85;
_PackTags.Command.Product[4].ProcessVariables[SEALTEMP].ID     := _PackTags.Command.Product[1].ProductID * 20 + 2;
_PackTags.Command.Product[4].ProcessVariables[SEALTEMP].Name   := 'Sealing Temp';
_PackTags.Command.Product[4].ProcessVariables[SEALTEMP].Unit   := 'C';
_PackTags.Command.Product[4].ProcessVariables[SEALTEMP].Value  := 95;
_PackTags.Command.Product[4].ProcessVariables[SEALTIME].ID     := _PackTags.Command.Product[1].ProductID * 20 + 3;
_PackTags.Command.Product[4].ProcessVariables[SEALTIME].Name   := 'Sealing Time';
_PackTags.Command.Product[4].ProcessVariables[SEALTIME].Unit   := 'ms';
_PackTags.Command.Product[4].ProcessVariables[SEALTIME].Value  := 80;
_PackTags.Command.Product[4].ProcessVariables[PULLWHEELS_VEL].ID    := _PackTags.Command.Product[1].ProductID * 20 + 4;
_PackTags.Command.Product[4].ProcessVariables[PULLWHEELS_VEL].Name  := 'Pull Wheels Vel';
_PackTags.Command.Product[4].ProcessVariables[PULLWHEELS_VEL].Unit  := 'mm/s';
_PackTags.Command.Product[4].ProcessVariables[PULLWHEELS_VEL].Value := 100;
_PackTags.Command.Product[4].ProcessVariables[PULLWHEELS_ACC].ID    := _PackTags.Command.Product[1].ProductID * 20 + 5;
_PackTags.Command.Product[4].ProcessVariables[PULLWHEELS_ACC].Name  := 'Pull Wheels Acc';
_PackTags.Command.Product[4].ProcessVariables[PULLWHEELS_ACC].Unit  := 'mm/s2';
_PackTags.Command.Product[4].ProcessVariables[PULLWHEELS_ACC].Value := 1000;
_PackTags.Command.Product[4].ProcessVariables[OPEN_POS].ID          := _PackTags.Command.Product[1].ProductID * 20 + 6;
_PackTags.Command.Product[4].ProcessVariables[OPEN_POS].Name        := 'Sealer Open Position';
_PackTags.Command.Product[4].ProcessVariables[OPEN_POS].Unit        := 'mm';
_PackTags.Command.Product[4].ProcessVariables[OPEN_POS].Value       := 105;
_PackTags.Command.Product[4].ProcessVariables[CLOSED_POS].ID        := _PackTags.Command.Product[1].ProductID * 20 + 7;
_PackTags.Command.Product[4].ProcessVariables[CLOSED_POS].Name      := 'Sealer Closed Position';
_PackTags.Command.Product[4].ProcessVariables[CLOSED_POS].Unit      := 'mm';
_PackTags.Command.Product[4].ProcessVariables[CLOSED_POS].Value     := 250;
_PackTags.Command.Product[4].ProcessVariables[SEALER_VEL].ID        := _PackTags.Command.Product[1].ProductID * 20 + 8;
_PackTags.Command.Product[4].ProcessVariables[SEALER_VEL].Name      := 'Sealer Vel';
_PackTags.Command.Product[4].ProcessVariables[SEALER_VEL].Unit      := 'mm/s';
_PackTags.Command.Product[4].ProcessVariables[SEALER_VEL].Value     := 100;
_PackTags.Command.Product[4].ProcessVariables[SEALER_ACC].ID        := _PackTags.Command.Product[1].ProductID * 20 + 9;
_PackTags.Command.Product[4].ProcessVariables[SEALER_ACC].Name      := 'Sealer Acc';
_PackTags.Command.Product[4].ProcessVariables[SEALER_ACC].Unit      := 'mm/s2';
_PackTags.Command.Product[4].ProcessVariables[SEALER_ACC].Value     := 1000;
_PackTags.Command.Product[4].ProcessVariables[UNWIND_VEL].ID        := _PackTags.Command.Product[1].ProductID * 20 + 10;
_PackTags.Command.Product[4].ProcessVariables[UNWIND_VEL].Name      := 'Unwind Vel';
_PackTags.Command.Product[4].ProcessVariables[UNWIND_VEL].Unit      := 'mm/s';
_PackTags.Command.Product[4].ProcessVariables[UNWIND_VEL].Value     := 100;
_PackTags.Command.Product[4].ProcessVariables[UNWIND_ACC].ID        := _PackTags.Command.Product[1].ProductID * 20 + 11;
_PackTags.Command.Product[4].ProcessVariables[UNWIND_ACC].Name      := 'Unwind Acc';
_PackTags.Command.Product[4].ProcessVariables[UNWIND_ACC].Unit      := 'mm/s2';
_PackTags.Command.Product[4].ProcessVariables[UNWIND_ACC].Value     := 1000;

//Product 5
_PackTags.Command.Product[5].ProductID                         := 522;
_PackTags.Command.Product[5].Ingredients[1].IngredientID       := 1;
_PackTags.Command.Product[5].Ingredients[1].Parameter[1].ID    := _PackTags.Command.Product[1].ProductID * 10 + 1;
_PackTags.Command.Product[5].Ingredients[1].Parameter[1].Name  := 'Material Type';
_PackTags.Command.Product[5].Ingredients[1].Parameter[1].Unit  := 'n/a';
_PackTags.Command.Product[5].Ingredients[1].Parameter[1].Value := 2;
_PackTags.Command.Product[5].Ingredients[1].Parameter[2].ID    := _PackTags.Command.Product[1].ProductID * 10 + 2;
_PackTags.Command.Product[5].Ingredients[1].Parameter[2].Name  := 'Material Thickness';
_PackTags.Command.Product[5].Ingredients[1].Parameter[2].Unit  := 'um';
_PackTags.Command.Product[5].Ingredients[1].Parameter[2].Value := 520;
_PackTags.Command.Product[5].ProcessVariables[LENGTH].ID       := _PackTags.Command.Product[1].ProductID * 20 + 1;
_PackTags.Command.Product[5].ProcessVariables[LENGTH].Name     := 'Length';
_PackTags.Command.Product[5].ProcessVariables[LENGTH].Unit     := 'mm';
_PackTags.Command.Product[5].ProcessVariables[LENGTH].Value    := 200;
_PackTags.Command.Product[5].ProcessVariables[SEALTEMP].ID     := _PackTags.Command.Product[1].ProductID * 20 + 2;
_PackTags.Command.Product[5].ProcessVariables[SEALTEMP].Name   := 'Sealing Temp';
_PackTags.Command.Product[5].ProcessVariables[SEALTEMP].Unit   := 'C';
_PackTags.Command.Product[5].ProcessVariables[SEALTEMP].Value  := 130;
_PackTags.Command.Product[5].ProcessVariables[SEALTIME].ID     := _PackTags.Command.Product[1].ProductID * 20 + 3;
_PackTags.Command.Product[5].ProcessVariables[SEALTIME].Name   := 'Sealing Time';
_PackTags.Command.Product[5].ProcessVariables[SEALTIME].Unit   := 'ms';
_PackTags.Command.Product[5].ProcessVariables[SEALTIME].Value  := 200;
_PackTags.Command.Product[5].ProcessVariables[PULLWHEELS_VEL].ID    := _PackTags.Command.Product[1].ProductID * 20 + 4;
_PackTags.Command.Product[5].ProcessVariables[PULLWHEELS_VEL].Name  := 'Pull Wheels Vel';
_PackTags.Command.Product[5].ProcessVariables[PULLWHEELS_VEL].Unit  := 'mm/s';
_PackTags.Command.Product[5].ProcessVariables[PULLWHEELS_VEL].Value := 100;
_PackTags.Command.Product[5].ProcessVariables[PULLWHEELS_ACC].ID    := _PackTags.Command.Product[1].ProductID * 20 + 5;
_PackTags.Command.Product[5].ProcessVariables[PULLWHEELS_ACC].Name  := 'Pull Wheels Acc';
_PackTags.Command.Product[5].ProcessVariables[PULLWHEELS_ACC].Unit  := 'mm/s2';
_PackTags.Command.Product[5].ProcessVariables[PULLWHEELS_ACC].Value := 1000;
_PackTags.Command.Product[5].ProcessVariables[OPEN_POS].ID          := _PackTags.Command.Product[1].ProductID * 20 + 6;
_PackTags.Command.Product[5].ProcessVariables[OPEN_POS].Name        := 'Sealer Open Position';
_PackTags.Command.Product[5].ProcessVariables[OPEN_POS].Unit        := 'mm';
_PackTags.Command.Product[5].ProcessVariables[OPEN_POS].Value       := 105;
_PackTags.Command.Product[5].ProcessVariables[CLOSED_POS].ID        := _PackTags.Command.Product[1].ProductID * 20 + 7;
_PackTags.Command.Product[5].ProcessVariables[CLOSED_POS].Name      := 'Sealer Closed Position';
_PackTags.Command.Product[5].ProcessVariables[CLOSED_POS].Unit      := 'mm';
_PackTags.Command.Product[5].ProcessVariables[CLOSED_POS].Value     := 250;
_PackTags.Command.Product[5].ProcessVariables[SEALER_VEL].ID        := _PackTags.Command.Product[1].ProductID * 20 + 8;
_PackTags.Command.Product[5].ProcessVariables[SEALER_VEL].Name      := 'Sealer Vel';
_PackTags.Command.Product[5].ProcessVariables[SEALER_VEL].Unit      := 'mm/s';
_PackTags.Command.Product[5].ProcessVariables[SEALER_VEL].Value     := 100;
_PackTags.Command.Product[5].ProcessVariables[SEALER_ACC].ID        := _PackTags.Command.Product[1].ProductID * 20 + 9;
_PackTags.Command.Product[5].ProcessVariables[SEALER_ACC].Name      := 'Sealer Acc';
_PackTags.Command.Product[5].ProcessVariables[SEALER_ACC].Unit      := 'mm/s2';
_PackTags.Command.Product[5].ProcessVariables[SEALER_ACC].Value     := 1000;
_PackTags.Command.Product[5].ProcessVariables[UNWIND_VEL].ID        := _PackTags.Command.Product[1].ProductID * 20 + 10;
_PackTags.Command.Product[5].ProcessVariables[UNWIND_VEL].Name      := 'Unwind Vel';
_PackTags.Command.Product[5].ProcessVariables[UNWIND_VEL].Unit      := 'mm/s';
_PackTags.Command.Product[5].ProcessVariables[UNWIND_VEL].Value     := 100;
_PackTags.Command.Product[5].ProcessVariables[UNWIND_ACC].ID        := _PackTags.Command.Product[1].ProductID * 20 + 11;
_PackTags.Command.Product[5].ProcessVariables[UNWIND_ACC].Name      := 'Unwind Acc';
_PackTags.Command.Product[5].ProcessVariables[UNWIND_ACC].Unit      := 'mm/s2';
_PackTags.Command.Product[5].ProcessVariables[UNWIND_ACC].Value     := 1000;


CurrentRecipeName := 'From PackTags';
END_METHOD

PROPERTY PUBLIC PackTags : ST_PackMLv30Ext
GET
PackTags := _packTags;
END_GET
END_PROPERTY

METHOD RaiseAlarm2Args
VAR_IN_OUT
    Alarm : FB_TcAlarm; //Alarm to be raised
END_VAR

VAR_INPUT
    String_1 : STRING; //First String Parameter (The Name of this component will be applied first automatically)
    String_2 : STRING; //Second String Parameter
END_VAR
F_RaiseAlarmWithStringParameters(Alarm    := Alarm,
                                 String_1 := Name,
                                 String_2 := String_1,
                                 String_3 := String_2);
END_METHOD

METHOD PROTECTED Resetting
VAR_INPUT
END_VAR
CASE _CurrentMode OF
    //=================================PRODUCTION MODE==================================
    E_PMLUnitMode.ePMLUnitMode_Production:
        IF DataFromPackML THEN
            product           := LREAL_TO_INT(_PackTags.Command.Parameter[2].Value);
            PullWheels.Length := _PackTags.Command.Product[product].ProcessVariables[LENGTH].Value;
			PullWheels.Velocity := _PackTags.Command.Product[product].ProcessVariables[PULLWHEELS_VEL].Value;
			PullWheels.Acceleration := _PackTags.Command.Product[product].ProcessVariables[PULLWHEELS_ACC].Value;
            Sealer.SealTime   := _PackTags.Command.Product[product].ProcessVariables[SEALTIME].Value;
            Sealer.Temp       := _PackTags.Command.Product[product].ProcessVariables[SEALTEMP].Value;
			Sealer.OpenPos := _PackTags.Command.Product[product].ProcessVariables[OPEN_POS].Value;
			Sealer.ClosedPos := _PackTags.Command.Product[product].ProcessVariables[CLOSED_POS].Value;
			Sealer.Velocity := _PackTags.Command.Product[product].ProcessVariables[SEALER_VEL].Value;
			Sealer.Acceleration := _PackTags.Command.Product[product].ProcessVariables[SEALER_ACC].Value;
			Unwind.Velocity := _PackTags.Command.Product[product].ProcessVariables[UNWIND_VEL].Value;
			Unwind.Acceleration := _PackTags.Command.Product[product].ProcessVariables[UNWIND_ACC].Value;
        END_IF

    E_PMLUnitMode.ePMLUnitMode_Maintenance, E_PMLUnitMode.ePMLUnitMode_Manual:
        ;
END_CASE

SUPER^.Resetting();
END_METHOD

METHOD PROTECTED Starting
VAR_INPUT
END_VAR
CASE _CurrentMode OF
    //=================================PRODUCTION MODE==================================
    E_PMLUnitMode.ePMLUnitMode_Production:
        // The seal bar can go to Execute, the others will be run in Mahcine Execute
        Sealer.Heat := TRUE;
        StateComplete();
    E_PMLUnitMode.ePMLUnitMode_Maintenance, E_PMLUnitMode.ePMLUnitMode_Manual:
        SUPER^.Starting();
END_CASE
END_METHOD

METHOD PROTECTED SubModuleMonitor : BOOL
VAR
    AlarmResponses : ARRAY[0..4] OF E_AlarmResponse; //Temporary response array	
END_VAR
// Check the sub Modules for Alarm Severity
SUPER^.SubModuleMonitor();

//Check the alarms at the machine level
_CurrentAlarmSeverity := F_GetMaxSeverityRaised(Alarms := MachineAlarms, CurrentSeverity := _CurrentAlarmSeverity);

//Check the severity of the machine level alarms
IF _CurrentState <> E_PMLState.ePMLState_Aborted AND _CurrentState <> E_PMLState.ePMLState_Aborting AND _CurrentState <> E_PMLState.ePMLState_Clearing AND
   _CurrentState <> E_PMLState.ePMLState_Stopped AND _CurrentState <> E_PMLState.ePMLState_Stopping THEN
    AlarmResponses := _ParentFaultResponseDefinitions;
    CASE AlarmResponses[CurrentAlarmSeverity] OF
        E_AlarmResponse.Abort_ImmediateError:
            AbortImmediateError(Name, TRUE);
        E_AlarmResponse.Abort_Immediate:
            AbortImmediate();
        E_AlarmResponse.Stop_Immediate:
            StopImmediate();
        E_AlarmResponse.Stop_Controlled:
            StopControlled();
        E_AlarmResponse.Hold_Immediate:
            HoldImmediate();
        E_AlarmResponse.Suspend_Immediate:
            SuspendImmediate();
        E_AlarmResponse.Suspend_Controlled:
            SuspendControlled();
        E_AlarmResponse.NoResponse:
            ;
    END_CASE
ELSIF _CurrentState = E_PMLState.ePMLState_Stopped OR _CurrentState = E_PMLState.ePMLState_Stopping THEN
    AlarmResponses := _ParentFaultResponseDefinitions;
    CASE AlarmResponses[CurrentAlarmSeverity] OF
        E_AlarmResponse.Abort_ImmediateError:
            AbortImmediateError(Name, TRUE);
        E_AlarmResponse.Abort_Immediate:
            AbortImmediate();
        E_AlarmResponse.NoResponse:
            ;
    END_CASE
END_IF
END_METHOD

METHOD PROTECTED Suspended
VAR_INPUT
END_VAR
IF THIS^.Sealer.sealbar.InTempRange THEN
	ChangeState(E_PMLCommand.ePMLCommand_Unsuspend);
END_IF
END_METHOD

METHOD PROTECTED Suspending
VAR_INPUT
END_VAR
CASE _CurrentMode OF
    //=================================PRODUCTION MODE==================================
    E_PMLUnitMode.ePMLUnitMode_Production:
        IF (Sealer.CurrentState = E_PMLState.ePMLState_Complete OR Sealer.CurrentState = E_PMLState.ePMLState_Idle) AND
           (PullWheels.CurrentState = E_PMLState.ePMLState_Complete OR PullWheels.CurrentState = E_PMLState.ePMLState_Idle) THEN
            StateComplete();
        END_IF
    E_PMLUnitMode.ePMLUnitMode_Maintenance, E_PMLUnitMode.ePMLUnitMode_Manual:
        SUPER^.Suspending();
END_CASE
END_METHOD

METHOD PROTECTED Unholding
VAR_INPUT
END_VAR
CASE _CurrentMode OF
    //=================================PRODUCTION MODE==================================
    E_PMLUnitMode.ePMLUnitMode_Production:
        StateComplete();
    E_PMLUnitMode.ePMLUnitMode_Maintenance, E_PMLUnitMode.ePMLUnitMode_Manual:
        SUPER^.Unholding();
END_CASE
END_METHOD

METHOD PROTECTED Unsuspending
VAR_INPUT
END_VAR
CASE _CurrentMode OF
    //=================================PRODUCTION MODE==================================
    E_PMLUnitMode.ePMLUnitMode_Production:
        StateComplete();
    E_PMLUnitMode.ePMLUnitMode_Maintenance, E_PMLUnitMode.ePMLUnitMode_Manual:
        SUPER^.Unsuspending();
END_CASE
END_METHOD

METHOD UpdateModeTimers
VAR
    currentTime  : T_DCTIME64;
    timeToUpdate : LREAL;
END_VAR

VAR_INST
    lastTime  : T_DCTIME64 := F_GetActualDcTime64();
    lastState : DINT;
    lastMode  : DINT;
END_VAR
IF _PackTags.Status.StateCurrent <> lastState THEN
    MEMSET(ADR(_PackTags.Admin.StateCurrentTime), 0, SIZEOF(_PackTags.Admin.StateCurrentTime));
    lastState := _PackTags.Status.StateCurrent;
END_IF

IF _PackTags.Status.UnitModeCurrent <> lastMode THEN
    MEMSET(ADR(_PackTags.Admin.ModeCurrentTime), 0, SIZEOF(_PackTags.Admin.ModeCurrentTime));
    lastMode := _PackTags.Status.UnitModeCurrent;
END_IF

currentTime := F_GetActualDcTime64();
IF lastTime <> 0 THEN
    timeToUpdate := ULINT_TO_LREAL(currentTime - lastTime) / 1_000_000_000.0;
END_IF

// only seconds get added to the cumulative timers 
IF timeToUpdate > 1 THEN
    _PackTags.Admin.ModeCummulativeTime[_PackTags.Status.UnitModeCurrent] := _PackTags.Admin.ModeCummulativeTime[_PackTags.Status.UnitModeCurrent] + LREAL_TO_DINT(timeToUpdate);
    _PackTags.Admin.ModeCurrentTime[_PackTags.Status.UnitModeCurrent]     := _PackTags.Admin.ModeCurrentTime[_PackTags.Status.UnitModeCurrent] + LREAL_TO_DINT(timeToUpdate);
    _PackTags.Admin.StateCummulativeTime[_PackTags.Status.UnitModeCurrent, _PackTags.Status.StateCurrent]
        := _PackTags.Admin.StateCummulativeTime[_PackTags.Status.UnitModeCurrent, _PackTags.Status.StateCurrent] + LREAL_TO_DINT(timeToUpdate);

    _PackTags.Admin.StateCurrentTime[_PackTags.Status.UnitModeCurrent, _PackTags.Status.StateCurrent] :=
        _PackTags.Admin.StateCurrentTime[_PackTags.Status.UnitModeCurrent, _PackTags.Status.StateCurrent] + LREAL_TO_DINT(timeToUpdate);

    lastTime := currentTime;
END_IF
END_METHOD

END_FUNCTION_BLOCK

// ---- Machine/HMI Connections/FB_ControlSource_HMI_Machine.TcPOU
FUNCTION_BLOCK FB_ControlSource_HMI_Machine EXTENDS FB_ControlSource_HMI
VAR_INPUT
END_VAR
VAR_OUTPUT
END_VAR
VAR
END_VAR

METHOD CyclicLogic
VAR_INPUT
END_VAR
SUPER^.CyclicLogic();

//Change the start permissive for the Machine 
MainPMLControl_Simplified.StartPermissive :=
    MainPMLControl_Standard.CurrentState = Tc3_PackML_V2.E_PMLState.ePMLState_Idle OR
    (MainPMLControl_Standard.CurrentState = Tc3_PackML_V2.E_PMLState.ePMLState_Held AND
    MAIN.ApicoSeed.Unwind.CurrentState = E_PMLState.ePMLState_Idle);
END_METHOD

END_FUNCTION_BLOCK

// ---- MAIN.TcPOU
PROGRAM MAIN
VAR
    ControlSource_HMI : FB_ControlSource_HMI_Machine;
    ApicoSeed          : FB_Machine := (Name := 'Apico_Seed');
    InitComplete      : BOOL;

    //Debug testing Recipe manager
    Value1 : INT;
    Value2 : INT;
END_VAR

CyclicLogic();

METHOD CyclicLogic
VAR_INPUT
END_VAR
IF NOT InitComplete THEN
    InitComplete := Initialize();
    RETURN;
END_IF

//Machine support HMI & Production Monitor
ControlSource_HMI.CyclicLogic();

//Machine Cyclic Logic
ApicoSeed.CyclicLogic();
END_METHOD

METHOD Initialize : BOOL
VAR_INPUT
END_VAR
//Top level machine initialization should happen here, in the main initialization method. Each subsequent "layer" of modules will be named within their respective "parent" intialize method
_AppInfo.KeepOutputsOnBP := TRUE;
IF NOT ControlSource_HMI.Registered THEN
    ApicoSeed.RegisterExternalController(ControlSource_HMI);
END_IF

ControlSource_HMI.CyclicLogic();
Initialize := TRUE;
END_METHOD

END_PROGRAM

// ---- GlobalTextList.TcGTLO
TEXTLIST GlobalTextList
  733 = '%0.1f °'
  282 = '%d'
  685 = '%s'
  680 = 'Abort'
  452 = 'Clear'
  809 = 'Clear Unwind'
  424 = 'EStop'
  744 = 'Hold'
  194 = 'ID:'
  517 = 'Kurwa Jebana'
  347 = 'MACHINE'
  46 = 'Maintenance'
  904 = 'Manual'
  929 = 'Production'
  181 = 'Reset'
  538 = 'Reset Unwind'
  206 = 'Simulate \nAll'
  436 = 'Simulate All'
  77 = 'Start'
  804 = 'Start Unwind'
  963 = 'State: %d'
  516 = 'State: %s'
  828 = 'Stop'
  806 = 'Suspend'
  995 = 'Temp Setpoint'
  197 = 'Unhold'
  832 = 'Unsuspend'
END_TEXTLIST

// ---- Machine/VISUs/V_Main.TcVIS
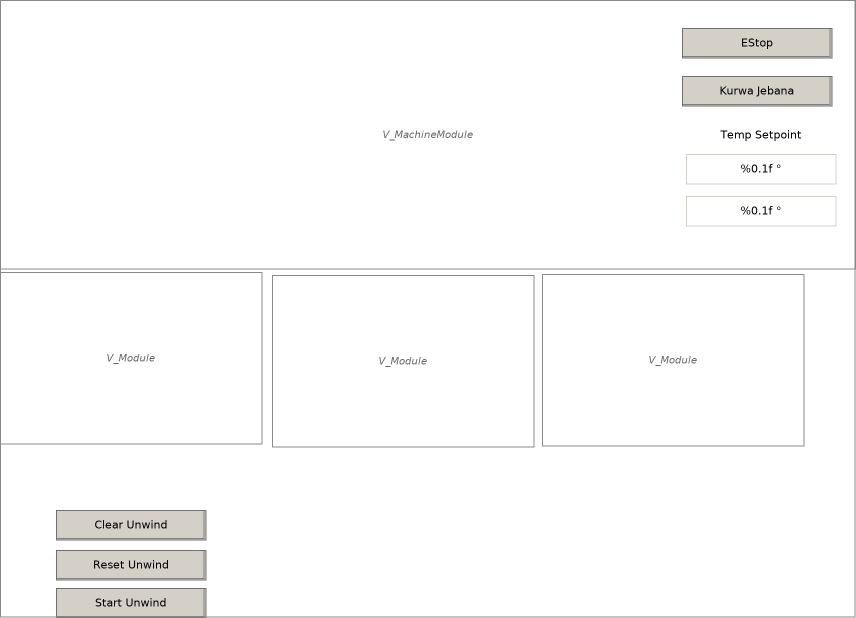
VISUALIZATION V_Main  // 856x618
    Frame (0,0 856x269)
        shows V_MachineModule(HMI := MAIN.ApicoSeed.PackMLBaseModule_HMI)
    Frame (0,272 262x172)
        shows V_Module(HMI := MAIN.ApicoSeed.PullWheels.PackMLBaseModule_HMI)
    Frame (272,275 262x172)
        shows V_Module(HMI := MAIN.ApicoSeed.Sealer.PackMLBaseModule_HMI)
    Frame (542,274 262x172)
        shows V_Module(HMI := MAIN.ApicoSeed.Unwind.PackMLBaseModule_HMI)
    Button (682,28 150x30), "EStop"
        toggle MAIN.ApicoSeed.EstopInput
    Button (682,76 150x30), "Kurwa Jebana"
        toggle MAIN.ApicoSeed.KurwaJebanaInput
    Textfield (686,154 150x30), "%0.1f °", text variable: MAIN.ApicoSeed.Sealer.SealBar._SetTemperature
        OnMouseDown: write the text variable via VisuDialogs.Numpad, min 20, max 400, title 'Sealer Bar Temp Setpoint', format %0.1f
    Label (686,120 150x30), "Temp Setpoint"
    Textfield (686,196 150x30), "%0.1f °", text variable: MAIN.ApicoSeed.Sealer.SealBar._ActualTemperature
    Button (56,510 150x30), "Clear Unwind"
        OnMouseClick: execute { MAIN.ApicoSeed.unwind.PackMLBaseModule_HMI.Command.State := E_PMLCommand.ePMLCommand_Clear; }
    Button (56,550 150x30), "Reset Unwind"
        OnMouseClick: execute { MAIN.ApicoSeed.unwind.PackMLBaseModule_HMI.Command.State := E_PMLCommand.ePMLCommand_Reset; }
    Button (56,588 150x30), "Start Unwind"
        OnMouseClick: execute { MAIN.ApicoSeed.unwind.PackMLBaseModule_HMI.Command.State := E_PMLCommand.ePMLCommand_Start; }
END_VISUALIZATION
